// TIA Portal V17 export
// export: Created 2024-09-27T18:48:47.5403244Z, ExportSetting WithDefaults, DisplayName Totally Integrated Automation Portal, DisplayVersion V17, DisplayName TIA Portal Openness, DisplayVersion V17, DisplayName TIA Portal Version Control Interface, DisplayVersion V17, DisplayName STEP 7 Professional, DisplayVersion V17, DisplayName STEP 7 Safety, DisplayVersion V17, DisplayName WinCC Professional, DisplayVersion V17
DATA_BLOCK "MC_Home_DB"   // DB11
// stored: AutoNumber true, DBAccessibleFromOPCUA true, InstanceOfName MC_Home, OfSystemLibElement MC_Home, OfSystemLibVersion 8.0
"MC_Home"
   // VAR_INPUT
   //    Axis : TO_Axis;
   //    Execute : Bool;
   //    Position : Real;
   //    Mode : Int;
   // END_VAR
   // VAR_OUTPUT
   //    Done : Bool;
   //    Busy : Bool;
   //    CommandAborted : Bool;
   //    Error : Bool;
   //    ErrorID : Word;
   //    ErrorInfo : Word;
   //    ReferenceMarkPosition : Real;
   // END_VAR
   // VAR
   //    FB_ID : DInt;
   // END_VAR
BEGIN
END_DATA_BLOCK
